Staubli VAL3: velOverwrite.pgx

public program velOverwrite(bool x_bOverwriteVel)
begin

  gotoxy(scMonitor, 0,5)
  put(scMonitor, "Velocity overwrite:")
  gotoxy(scMonitor, 20,5)
  if(x_bOverwriteVel == true)
    put(scMonitor, "enabled")
  else
    put(scMonitor, "disabled")
  endIf

end
